PROGRAM MAIN
VAR
END_VAR

// Niet gemaakt

(*
Personeelsdata in visu

Creëer of overschrijf personeelsdata vanuit de visualisatie in de arrays. 
Pas hierbij de checker functions toe om de leeftijd de beperken van 0 tot 100 jaar. 
Gender doe je via een enum.
*)

END_PROGRAM

(* stored: Version 1.1.0.1, ProductVersion 3.1.4024.12
   POU MAIN: Id {56ba40b1-245e-4afd-9610-dc0c429edfb0}, SpecialFunc None *)
